FUNCTION AccelerometerReadings : BOOL
VAR_INPUT
	q : ARRAY [0..2] OF LREAL;
	qdot : ARRAY [0..2] OF LREAL;
	qddot : ARRAY [0..2] OF LREAL;
	L : ARRAY [0..2] OF LREAL;
	Tip_to_IMU : REFERENCE TO ARRAY [0..2] OF FB_Vector3;
	AccelerometerReadingsOut : REFERENCE TO ARRAY [0..2] OF FB_Vector3;
	gravity_vector : REFERENCE TO FB_Vector3;
	
END_VAR
VAR
	
	z0 : FB_Vector3 := (X := 0, Y := 0, Z := 1);
	
	T_from_i_1_to_i : FB_Matrix4x4;
	Rot : FB_Matrix3x3;
	Rot_Trans : TransposeMatrixAccessor;
	Rot_IMU_Joint : FB_Matrix3x3;
	w : ARRAY [0..2] OF FB_Vector3;
	wdot : ARRAY [0..2] OF FB_Vector3;
	vdot : ARRAY [0..2] OF FB_Vector3;
	vIMUdot : ARRAY [0..2] OF FB_Vector3;	

	p : FB_Vector3; 

	i : USINT;
	
	
	prod_z0_qdot : FB_Vector3;	
	

	tmp : SubMatrixAccessor;
	
	prod_z0_qddot : FB_Vector3;	

		
		
	prod_Rottrans_grav : FB_Vector3;
	cross_wdot_p : FB_Vector3;
	cross_w_p : FB_Vector3;
	cross_w_w_p : FB_Vector3;
	
	cross_wdot_imu : FB_Vector3;
	cross_w_imu : FB_Vector3;
	cross_w_w_imu : FB_Vector3;

	sum_w_prod_z0_qdot : FB_Vector3;
	
	sum_wdot_prod_z0_qddot_cross_w_prod_z0_qdot : FB_Vector3;
	cross_w_prod_z0_qdot : FB_Vector3;
	
	prod_Rottrans_vdot : FB_Vector3;

	
	
	
END_VAR


//gravity_vector.SetI(0, 0);
//gravity_vector.SetI(1, 9.8*1);
//gravity_vector.SetI(2, 0);


//z0.SetI(0,0);
//z0.SetI(1,0);
//z0.SetI(2,1);

Rot_IMU_Joint.SetRC(0,0,0);
Rot_IMU_Joint.SetRC(0,1,0);
Rot_IMU_Joint.SetRC(0,2,1);
Rot_IMU_Joint.SetRC(1,0,1);
Rot_IMU_Joint.SetRC(1,1,0);
Rot_IMU_Joint.SetRC(1,2,0);
Rot_IMU_Joint.SetRC(2,0,0);
Rot_IMU_Joint.SetRC(2,1,1);
Rot_IMU_Joint.SetRC(2,2,0);

FOR i:=0 TO 2 DO
	
   	F_DH(theta:= q[i],d:=0,a:=L[i],alpha:=0,T_from_i_1_to_i);
	tmp := T_from_i_1_to_i.GetSubMatrixAccessor(RowStart:=0,RowCount:=3,ColStart:=0,ColCount:=3);
	tmp.CopyTo(Rot);
	Rot_Trans := Rot.GetTransposeMatrixAccessor();
	
	p.SetI(0,L[i]);
	p.SetI(1,0);
	p.SetI(2,0);
	
	IF i > 0 THEN
//        w(:, i) =  R'*(w(:, i-1) + z0.*qdot(i));
		z0.CopyTo(prod_z0_qdot); 								// z0.*qdot(i)
		prod_z0_qdot.Scale(qdot[i]);
		prod_z0_qdot.CopyTo(sum_w_prod_z0_qdot);
		sum_w_prod_z0_qdot.ElementSum(w[i-1]);
		Matrix_Product(Rot_Trans,sum_w_prod_z0_qdot,w[i]); 



//        wdot(:, i) = R'*(wdot(:, i-1) +  z0.*qddot(i) + ...
//            cross(w(:, i-1), z0.*qdot(i)));
		z0.CopyTo(prod_z0_qddot); 								
		prod_z0_qddot.Scale(qddot[i]);		
		F_Cross2(w[i-1],prod_z0_qdot,cross_w_prod_z0_qdot);	    
		
		wdot[i-1].CopyTo(sum_wdot_prod_z0_qddot_cross_w_prod_z0_qdot);
		sum_wdot_prod_z0_qddot_cross_w_prod_z0_qdot.ElementSum(prod_z0_qddot);
		sum_wdot_prod_z0_qddot_cross_w_prod_z0_qdot.ElementSum(cross_w_prod_z0_qdot);
		Matrix_Product(Rot_Trans,sum_wdot_prod_z0_qddot_cross_w_prod_z0_qdot,wdot[i]); 

//        vdot(:,i) = R'*vdot(:,i-1) + cross(wdot(:,i), p) + ...
//            cross(w(:,i), cross(w(:,i),p));-----------------------------------------------------------------
			
		Matrix_Product(Rot_Trans,vdot[i-1],prod_Rottrans_vdot); 				
		F_Cross2(wdot[i],p,cross_wdot_p);
		F_Cross2(w[i],p,cross_w_p);
		F_Cross2(w[i],cross_w_p,cross_w_w_p);
		
		prod_Rottrans_vdot.CopyTo(vdot[i]);
		vdot[i].ElementSum(cross_wdot_p);
		vdot[i].ElementSum(cross_w_w_p);
		
		

		
		


//        vIMUdot(:,i) = vdot(:,i) + cross(wdot(:,i),Tip_to_IMU(:,i)) + ...
//            cross(w(:,i),cross(w(:,i),Tip_to_IMU(:,i)));

		F_Cross2(wdot[i],Tip_to_IMU[i],cross_wdot_imu);
		F_Cross2(w[i],Tip_to_IMU[i],cross_w_imu);
		F_Cross2(w[i],cross_w_imu,cross_w_w_imu); //cross_w_p --> cross_w_imu 
		
		
		vdot[i].CopyTo(vIMUdot[i]);
		vIMUdot[i].ElementSum(cross_wdot_imu);
		vIMUdot[i].ElementSum(cross_w_w_imu);





	ELSE		
//		        w(:, i) =  R'*(z0.*qdot(i));
		z0.CopyTo(prod_z0_qdot); 								
		prod_z0_qdot.Scale(qdot[i]);
		Matrix_Product(Rot_Trans,prod_z0_qdot,w[i]); 

//        wdot(:, i) = R'*(z0.*qddot(i));
		z0.CopyTo(prod_z0_qddot); 								
		prod_z0_qddot.Scale(qddot[i]);									
		Matrix_Product(Rot_Trans,prod_z0_qddot,wdot[i]); // R'*(z0.*qddot(i));	


//        vdot(:,i) = R'*grav + cross(wdot(:,i), p) + ...
//            cross(w(:,i), cross(w(:,i),p));
		Matrix_Product(Rot_Trans,gravity_vector,prod_Rottrans_grav);
		F_Cross2(wdot[i],p,cross_wdot_p);
		F_Cross2(w[i],p,cross_w_p);
		F_Cross2(w[i],cross_w_p,cross_w_w_p);
		
		
		prod_Rottrans_grav.CopyTo(vdot[i]);
		vdot[i].ElementSum(cross_wdot_p);
		vdot[i].ElementSum(cross_w_w_p);


//        vIMUdot(:,i) = vdot(:,i) + cross(wdot(:,i),Tip_to_IMU(:,i)) + ...
//            cross(w(:,i),cross(w(:,i),Tip_to_IMU(:,i)));

		F_Cross2(wdot[i],Tip_to_IMU[i],cross_wdot_imu);
		F_Cross2(w[i],Tip_to_IMU[i],cross_w_imu);
		F_Cross2(w[i],cross_w_imu,cross_w_w_imu); //cross_w_p --> cross_w_imu 
		
		
		vdot[i].CopyTo(vIMUdot[i]);
		vIMUdot[i].ElementSum(cross_wdot_imu);
		vIMUdot[i].ElementSum(cross_w_w_imu);



	END_IF	
	Matrix_Product(Rot_IMU_Joint,vIMUdot[i],AccelerometerReadingsOut[i]);	
	
END_FOR;

END_FUNCTION

(* stored: Version 1.1.0.1, ProductVersion 3.1.4024.9
   POU AccelerometerReadings: Id {976375c1-9358-45cc-b0bb-504490b4c614}, SpecialFunc None *)
